Fanuc KAREL source: kb00072.KL

-- PROVISIONAL review KL for V940-1; original PC SHA256 a7736bb6cf8a708e4d671ec0405ee7cc8cdda82cfddbf2d36407b4a93a37232e
-- Incomplete behavior may be omitted. Consult companion uncertainty JSON. Do not deploy.
PROGRAM KB00072
%NOLOCKGROUP
BEGIN
  -- V9_ZERO_TABLE_METADATA_HINT layout=0002_ascii; no indexed target words; source/name/runtime held
  -- UNRESOLVED_PC offsets 5-14; opcodes 3F,75
  -- UNRESOLVED_PC offsets 19-26; opcodes 9D,23
  -- UNRESOLVED_PC offsets 31-38; opcodes 9D,23
  -- UNRESOLVED_PC offsets 43-50; opcodes 9D,23
  -- UNRESOLVED_PC offsets 55-62; opcodes 9D,23
  -- UNRESOLVED_PC offsets 67-109; opcodes 27,22,2A,22,22,22,22,22,31
  -- UNRESOLVED_PC offsets 114-118; opcodes 7F
END KB00072
